// TIA Portal V18 export
FUNCTION_BLOCK "Select_remote_or_auto"   // FB24, FBD
{ S7_Optimized_Access := 'TRUE' }
VERSION : 0.1
// stored: AutoNumber true, IsIECCheckEnabled false, IsRetainMemResEnabled false, MemoryReserve 100, SetENOAutomatically false, UDAEnableTagReadback false
BEGIN
END_FUNCTION_BLOCK
